// TIA Portal V19 export
VAR_GLOBAL   // PLC tag table "faceplate"
   "Start Button 0" AT %I0.0 : Bool;
   "Stop Button 0" AT %I0.1 : Bool;
   "Start Button 1" AT %I0.2 : Bool;
   "Stop Button 1" AT %I0.3 : Bool;
   "Start Button 2" AT %I0.4 : Bool;
   "Stop Button 2" AT %I0.5 : Bool;
   "Start Button 3" AT %I0.6 : Bool;
   "Stop Button 3" AT %I0.7 : Bool;
   "Belt Conveyor (4m) 0 (+)" AT %Q0.0 : Bool;
   "Belt Conveyor (4m) 0 (-)" AT %Q0.1 : Bool;
   "Belt Conveyor (4m) 1 (+)" AT %Q0.2 : Bool;
   "Belt Conveyor (4m) 1 (-)" AT %Q0.3 : Bool;
   "Belt Conveyor (4m) 2 (+)" AT %Q0.4 : Bool;
   "Belt Conveyor (4m) 2 (-)" AT %Q0.5 : Bool;
   "Belt Conveyor (4m) 3 (+)" AT %Q0.6 : Bool;
   "Belt Conveyor (4m) 3 (-)" AT %Q0.7 : Bool;
END_VAR
